PROGRAM MAIN
VAR
END_VAR

END_PROGRAM

(* stored: Version 1.1.0.1
   POU MAIN: Id {57b04bfc-bfd4-4571-98c2-d54fc671c159} *)
